// TwinCAT 3 PLC project bnct_plc
// ProgramVersion: 3.1.4024.0
// libraries:
//   Tc2_Standard, * (Beckhoff Automation GmbH)
//   Tc2_System, * (Beckhoff Automation GmbH)
//   Tc3_Module, * (Beckhoff Automation GmbH)
// project tree:
//   DUTs/ Call_Values_To_PC_Struct.TcDUT, Com_StripperEleMach_Struct.TcDUT, ST_FrameCmd.TcDUT
//   DUTs/Read_Status_Struct/ Read_AR_Values_To_PC_Struct.TcDUT, Read_BD_Values_To_PC_Struct.TcDUT, Read_BLPS1_Values_To_PC_Struct.TcDUT, Read_BLPS3_Values_To_PC_Struct.TcDUT, Read_BLVac1_Values_To_PC_Struct.TcDUT, Read_BLVac2_Values_To_PC_Struct.TcDUT, Read_BLVac3_Values_To_PC_Struct.TcDUT, Read_IL_Values_To_PC_Struct.TcDUT, Read_INJLPS_Values_To_PC_Struct.TcDUT, Read_ISPS_Values_To_PC_Struct.TcDUT, Read_ISVac_Values_To_PC_Struct.TcDUT, Read_MainPS_Values_To_PC_Struct.TcDUT, Read_MainVac_Values_To_PC_Struct.TcDUT, Read_RFG_Values_To_PC_Struct.TcDUT, Read_WC_Values_To_PC_Struct.TcDUT
//   DUTs/System_Status_Struct/ S_ARValues_To_PC_Struct.TcDUT, S_BDValues_To_PC_Struct.TcDUT, S_BLPS1Values_To_PC_Struct.TcDUT, S_BLPS3Values_To_PC_Struct.TcDUT, S_BLVac1Values_To_PC_Struct.TcDUT, S_BLVac2Values_To_PC_Struct.TcDUT, S_BLVac3Values_To_PC_Struct.TcDUT, S_ILValues_To_PC_Struct.TcDUT, S_INJLPSValues_To_PC_Struct.TcDUT, S_ISPSValues_To_PC_Struct.TcDUT, S_ISVacValues_To_PC_Struct.TcDUT, S_MainPSValues_To_PC_Struct.TcDUT, S_MainVacValues_To_PC_Struct.TcDUT, S_RFValues_To_PC_Struct.TcDUT, S_WCValues_To_PC_Struct.TcDUT, TCSSys_Struct.TcDUT
//   / PlcTask.TcTTO
//   POUs/ Call_Values_To_PC.TcPOU, Com_StripperEleMach.TcPOU, MAIN.TcPOU, GVL_TCSSys.TcPOU
// real-time tasks:
//   TASK PlcTask: cycle T#10ms, priority 20, ADS port 350

CONFIGURATION bnct_plc
    RESOURCE PLC ON TwinCAT3
        TASK PlcTask(INTERVAL := T#10ms, PRIORITY := 20);
        PROGRAM MAIN WITH PlcTask : MAIN;
        PROGRAM Call_Values_To_PC WITH PlcTask : Call_Values_To_PC;
        PROGRAM Com_StripperEleMach WITH PlcTask : Com_StripperEleMach;
        PROGRAM GVL_TCSSys WITH PlcTask : GVL_TCSSys;
    END_RESOURCE
END_CONFIGURATION

// ---- DUTs/Call_Values_To_PC_Struct.TcDUT
TYPE Call_Values_To_PC_Struct :
UNION
	Read_WC_Values_To_PC:READ_WC_Values_To_PC_Struct; //3.4.1水冷系统
	Read_AR_Values_To_PC:Read_AR_Values_To_PC_Struct; //3.4.2气动系统
	Read_ISVac_Values_To_PC:Read_ISVac_Values_To_PC_Struct; //3.4.3离子源真空系统
	Read_MainVac_Values_To_PC:Read_MainVac_Values_To_PC_Struct; //3.4.4主真空系统
	Read_BLVac1_Values_To_PC:Read_BLVac1_Values_To_PC_Struct; //3.4.5 束流线 1（公共束流线）真空系统
	Read_BLVac2_Values_To_PC:Read_BLVac2_Values_To_PC_Struct; //3.4.6 束流线 2（公共束流线）真空系统
	Read_BLVac3_Values_To_PC:Read_BLVac3_Values_To_PC_Struct; //3.4.7 束流线 3（公共束流线）真空系统
	Read_ISPS_Values_To_PC:Read_ISPS_Values_To_PC_Struct; //3.4.8 离子源电源系统 
	Read_INJLPS_Values_To_PC:Read_INJLPS_Values_To_PC_Struct; //3.4.9 注入线电源系统
	Read_MainPS_Values_To_PC:Read_MainPS_Values_To_PC_Struct;  //3.4.10 主器电源系统
	Read_BLPS1_Values_To_PC:Read_BLPS1_Values_To_PC_Struct; //3.4.11 束流线 1（公共束流线）电源系统
	Read_BLPS3_Values_To_PC:Read_BLPS3_Values_To_PC_Struct; //3.4.12 束流线 3（中子靶束流线）电源系统
	Read_RFG_Values_To_PC:Read_RFG_Values_To_PC_Struct; //3.4.13 高频系统
	Read_BD_Values_To_PC:Read_BD_Values_To_PC_Struct; //3.4.14 束流测量系统
	Read_IL_Values_To_PC:Read_IL_Values_To_PC_Struct; //3.4.15 联锁系统
END_UNION
END_TYPE

// ---- DUTs/Com_StripperEleMach_Struct.TcDUT
TYPE Com_StripperEleMach_Struct :
STRUCT
	Axis1_bEleMachinery_C_Power        : BOOL;
    Axis1_bEleMachinery_C_JF           : BOOL;
    Axis1_bEleMachinery_C_JB           : BOOL;
	Axis1_fEleMachinery_C_AbPos        : REAL;
    Axis1_fEleMachinery_C_AbPosVelo    : REAL;
    Axis1_bEleMachinery_C_AbPosExecute : BOOL;
    Axis1_bEleMachinery_C_Reset        : BOOL;
	Axis2_bEleMachinery_C_Power        : BOOL;
    Axis2_bEleMachinery_C_JF           : BOOL;
    Axis2_bEleMachinery_C_JB           : BOOL;
	Axis2_fEleMachinery_C_AbPos        : REAL;
    Axis2_fEleMachinery_C_AbPosVelo    : REAL;
    Axis2_bEleMachinery_C_AbPosExecute : BOOL;
    Axis2_bEleMachinery_C_Reset        : BOOL;
END_STRUCT
END_TYPE

// ---- DUTs/Read_Status_Struct/Read_AR_Values_To_PC_Struct.TcDUT
TYPE Read_AR_Values_To_PC_Struct :
UNION
	S_ARValues_To_PC:S_ARValues_To_PC_Struct;
END_UNION
END_TYPE

// ---- DUTs/Read_Status_Struct/Read_BD_Values_To_PC_Struct.TcDUT
TYPE Read_BD_Values_To_PC_Struct :
UNION
	S_BDValues_To_PC:S_BDValues_To_PC_Struct;
END_UNION
END_TYPE

// ---- DUTs/Read_Status_Struct/Read_BLPS1_Values_To_PC_Struct.TcDUT
TYPE Read_BLPS1_Values_To_PC_Struct :
UNION
	S_BLPS1Values_To_PC:S_BLPS1Values_To_PC_Struct;
END_UNION
END_TYPE

// ---- DUTs/Read_Status_Struct/Read_BLPS3_Values_To_PC_Struct.TcDUT
TYPE Read_BLPS3_Values_To_PC_Struct :
UNION
	S_BLPS3Values_To_PC:S_BLPS3Values_To_PC_Struct;
END_UNION
END_TYPE

// ---- DUTs/Read_Status_Struct/Read_BLVac1_Values_To_PC_Struct.TcDUT
TYPE Read_BLVac1_Values_To_PC_Struct :
UNION
	S_BLVac1Values_To_PC:S_BLVac1Values_To_PC_Struct;
END_UNION
END_TYPE

// ---- DUTs/Read_Status_Struct/Read_BLVac2_Values_To_PC_Struct.TcDUT
TYPE Read_BLVac2_Values_To_PC_Struct :
UNION
	S_BLVac2Values_To_PC:S_BLVac2Values_To_PC_Struct;
END_UNION
END_TYPE

// ---- DUTs/Read_Status_Struct/Read_BLVac3_Values_To_PC_Struct.TcDUT
TYPE Read_BLVac3_Values_To_PC_Struct :
UNION
	S_BLVac3Values_To_PC:S_BLVac3Values_To_PC_Struct;
END_UNION
END_TYPE

// ---- DUTs/Read_Status_Struct/Read_IL_Values_To_PC_Struct.TcDUT
TYPE Read_IL_Values_To_PC_Struct :
UNION
	S_ILValues_To_PC:S_ILValues_To_PC_Struct;
	// S_ILValues_To_PC:ARRAY[0..116]OF BYTE;
END_UNION
END_TYPE

// ---- DUTs/Read_Status_Struct/Read_INJLPS_Values_To_PC_Struct.TcDUT
TYPE Read_INJLPS_Values_To_PC_Struct :
UNION
	S_INJLPSValues_To_PC:S_INJLPSValues_To_PC_Struct;
END_UNION
END_TYPE

// ---- DUTs/Read_Status_Struct/Read_ISPS_Values_To_PC_Struct.TcDUT
TYPE Read_ISPS_Values_To_PC_Struct :
UNION
	S_ISPSValues_To_PC:S_ISPSValues_To_PC_Struct;
END_UNION
END_TYPE

// ---- DUTs/Read_Status_Struct/Read_ISVac_Values_To_PC_Struct.TcDUT
TYPE Read_ISVac_Values_To_PC_Struct :
UNION
	S_ISVacValues_To_PC:S_ISVacValues_To_PC_Struct;
END_UNION
END_TYPE

// ---- DUTs/Read_Status_Struct/Read_MainPS_Values_To_PC_Struct.TcDUT
TYPE Read_MainPS_Values_To_PC_Struct :
UNION
	S_MainPSValues_To_PC:S_MainPSValues_To_PC_Struct;
END_UNION
END_TYPE

// ---- DUTs/Read_Status_Struct/Read_MainVac_Values_To_PC_Struct.TcDUT
TYPE Read_MainVac_Values_To_PC_Struct :
UNION
	S_MainVacValues_To_PC:S_MainVacValues_To_PC_Struct;
END_UNION
END_TYPE

// ---- DUTs/Read_Status_Struct/Read_RFG_Values_To_PC_Struct.TcDUT
TYPE Read_RFG_Values_To_PC_Struct :
UNION
	S_RFValues_To_PC:S_RFValues_To_PC_Struct;
END_UNION
END_TYPE

// ---- DUTs/Read_Status_Struct/Read_WC_Values_To_PC_Struct.TcDUT
TYPE Read_WC_Values_To_PC_Struct :
UNION
	S_WCValues_To_PC:S_WCValues_To_PC_Struct;
END_UNION
END_TYPE

// ---- DUTs/System_Status_Struct/S_ARValues_To_PC_Struct.TcDUT
TYPE S_ARValues_To_PC_Struct :
STRUCT
	PARAM000:BOOL ; //注入线隔断阀开到位
	PARAM001:BOOL ; //注入线隔断阀关到位
	PARAM002:BOOL ; //注入线隔断阀正在开
	PARAM003:BOOL ; //注入线隔断阀正在关
	PARAM004:BOOL ; //注入线隔断阀开启操作错误
	PARAM005:BOOL ; //注入线隔断阀关闭操作错误
	PARAM006:BOOL ; //束流线隔断阀 1 开到位
	PARAM007:BOOL ; //束流线隔断阀 1 关到位
	PARAM008:BOOL ; //束流线隔断阀 1 正在开
	PARAM009:BOOL ; //束流线隔断阀 1 正在关
	PARAM010:BOOL ; //束流线隔断阀 1 开启操作错误
	PARAM011:BOOL ; //束流线隔断阀 1 关闭操作错误
	PARAM012:BOOL ; //束流线隔断阀 2 开到位
	PARAM013:BOOL ; //束流线隔断阀 2 关到位
	PARAM014:BOOL ; //束流线隔断阀 2 正在开
	PARAM015:BOOL ; //束流线隔断阀 2 正在关
	PARAM016:BOOL ; //束流线隔断阀 2 开启操作错误
	PARAM017:BOOL ; //束流线隔断阀 2 关闭操作错误
	PARAM018:BOOL ; //束流线隔断阀 3 开到位
	PARAM019:BOOL ; //束流线隔断阀 3 关到位
	PARAM020:BOOL ; //束流线隔断阀 3 正在开
	PARAM021:BOOL ; //束流线隔断阀 3 正在关
	PARAM022:BOOL ; //束流线隔断阀 3 开启操作错误
	PARAM023:BOOL ; //束流线隔断阀 3 关闭操作错误
	PARAM024:BOOL ; //注入线 FC 拉出到位
	PARAM025:BOOL ; //注入线 FC 插入到位
	PARAM026:BOOL ; //注入线 FC 正在拉出
	PARAM027:BOOL ; //注入线 FC 正在插入
	PARAM028:BOOL ; //注入线 FC 拉出操作错误
	PARAM029:BOOL ; //注入线 FC 插入操作错误
	PARAM030:BOOL ; //内靶拉出到位
	PARAM031:BOOL ; //内靶插入到位
	PARAM032:BOOL ; //内靶正在拉出
	PARAM033:BOOL ; //内靶正在插入
	PARAM034:BOOL ; //内靶拉出操作错误
	PARAM035:BOOL ; //内靶插入操作错误
	PARAM036:BOOL ; //引出 FC 拉出到位
	PARAM037:BOOL ; //引出 FC 插入到位
	PARAM038:BOOL ; //引出 FC 正在拉出
	PARAM039:BOOL ; //引出 FC 正在插入
	PARAM040:BOOL ; //引出 FC 拉出操作错误
	PARAM041:BOOL ; //引出 FC 插入操作错误
	PARAM042:BOOL ; //荧光靶 1 拉出到位
	PARAM043:BOOL ; //荧光靶 1 插入到位
	PARAM044:BOOL ; //荧光靶 1 正在拉出
	PARAM045:BOOL ; //荧光靶 1 正在插入
	PARAM046:BOOL ; //荧光靶 1 拉出操作错误
	PARAM047:BOOL ; //荧光靶 1 插入操作错误
	PARAM048:BOOL ; //荧光靶 2 拉出到位
	PARAM049:BOOL ; //荧光靶 2 插入到位
	PARAM050:BOOL ; //荧光靶 2 正在拉出
	PARAM051:BOOL ; //荧光靶 2 正在插入
	PARAM052:BOOL ; //荧光靶 2 拉出操作错误
	PARAM053:BOOL ; //荧光靶 2 插入操作错误
	PARAM054:BOOL ; //荧光靶 3 拉出到位
	PARAM055:BOOL ; //荧光靶 3 插入到位
	PARAM056:BOOL ; //荧光靶 3 正在拉出
	PARAM057:BOOL ; //荧光靶 3 正在插入
	PARAM058:BOOL ; //荧光靶 3 拉出操作错误
	PARAM059:BOOL ; //荧光靶 3 插入操作错误
	PARAM060:BOOL ; //双丝 1 拉出到位
	PARAM061:BOOL ; //双丝 1 插入到位
	PARAM062:BOOL ; //双丝 1 正在拉出
	PARAM063:BOOL ; //双丝 1 正在插入
	PARAM064:BOOL ; //双丝 1 拉出操作错误
	PARAM065:BOOL ; //双丝 1 插入操作错误
	PARAM066:BOOL ; //双丝 2 拉出到位
	PARAM067:BOOL ; //双丝 2 插入到位
	PARAM068:BOOL ; //双丝 2 正在拉出
	PARAM069:BOOL ; //双丝 2 正在插入
	PARAM070:BOOL ; //双丝 2 拉出操作错误
	PARAM071:BOOL ; //双丝 2 插入操作错误

END_STRUCT
END_TYPE

// ---- DUTs/System_Status_Struct/S_BDValues_To_PC_Struct.TcDUT
TYPE S_BDValues_To_PC_Struct :
STRUCT
	PARAM000:BOOL  ;// 剥离靶1电机使能指令 
	PARAM001:BOOL  ;// 剥离靶1电机绝对运动触发指令 
	PARAM002:REAL  ;// 剥离靶1电机绝对运动位置指令 
	PARAM003:REAL  ;// 剥离靶1电机绝对运动速度指令 
	PARAM004:BOOL  ;// 剥离靶1电机复位指令 
	PARAM005:BOOL  ;// 剥离靶1电机JOG前进指令 
	PARAM006:BOOL  ;// 剥离靶1电机JOG后退指令 
	PARAM007:BOOL  ;// 剥离靶1电机急停指令 
	PARAM008:BOOL  ;// 剥离靶1电机绝对运动完成 
	PARAM009:BOOL  ;// 剥离靶1电机绝对运动正在进行 
	PARAM010:REAL  ;// 剥离靶1电机位置状态 
	PARAM011:REAL  ;// 剥离靶1电机速度状态 
	PARAM012:BOOL  ;// 剥离靶1电机JOG运动完成 
	PARAM013:BOOL  ;// 剥离靶1电机JOG运动正在进行 
	PARAM014:UDINT ;// 剥离靶1电机故障编码 
	PARAM015:INT   ;// 剥离靶1电位器位置 
	PARAM016:BOOL  ;// 剥离靶2电机使能指令 
	PARAM017:BOOL  ;// 剥离靶2电机绝对运动触发指令 
	PARAM018:REAL  ;// 剥离靶2电机绝对运动位置指令 
	PARAM019:REAL  ;// 剥离靶2电机绝对运动速度指令 
	PARAM020:BOOL  ;// 剥离靶2电机复位指令 
	PARAM021:BOOL  ;// 剥离靶2电机JOG前进指令 
	PARAM022:BOOL  ;// 剥离靶2电机JOG后退指令 
	PARAM023:BOOL  ;// 剥离靶2电机急停指令 
	PARAM024:BOOL  ;// 剥离靶2电机绝对运动完成 
	PARAM025:BOOL  ;// 剥离靶2电机绝对运动正在进行 
	PARAM026:REAL  ;// 剥离靶2电机位置 
	PARAM027:REAL  ;// 剥离靶2电机速度 
	PARAM028:BOOL  ;// 剥离靶2电机JOG运动完成 
	PARAM029:BOOL  ;// 剥离靶2电机JOG运动正在进行 
	PARAM030:UDINT ;// 剥离靶2电机故障编码
	PARAM031:INT   ;// 剥离靶2电位器位置 
	PARAM032:REAL  ;// 束流通道1（mA）：注入FC 
	PARAM033:REAL  ;// 束流通道2（mA）:内靶 
	PARAM034:REAL  ;// 束流通道3（mA）：剥离靶 
	PARAM035:REAL  ;// 束流通道4（mA）：引出FC 
	PARAM036:REAL  ;// 束流通道5（mA）：铍靶 
	PARAM037:REAL  ;// 束流通道6（uA）：备用1 
	PARAM038:REAL  ;// 束流通道7（uA）：备用2 
	PARAM039:REAL  ;// 束流通道8（mA）：备用3 
	PARAM040:REAL  ;// 束流通道9（uA）：光阑1-上 
	PARAM041:REAL  ;// 束流通道10（uA）：光阑2-上 
	PARAM042:REAL  ;// 束流通道11（uA）：光阑1-下 
	PARAM043:REAL  ;// 束流通道12（uA）：光阑2-下 
	PARAM044:REAL  ;// 束流通道13（uA）：光阑1-左 
	PARAM045:REAL  ;// 束流通道14（uA）：光阑2-左 
	PARAM046:REAL  ;// 束流通道15（uA）：光阑1-右 
	PARAM047:REAL  ;// 束流通道16（uA）：光阑2-右 
END_STRUCT
END_TYPE

// ---- DUTs/System_Status_Struct/S_BLPS1Values_To_PC_Struct.TcDUT
TYPE S_BLPS1Values_To_PC_Struct :
STRUCT
	PARAM000:BOOL ; //  束流线1电源自动运行，TRUE为开启 
	PARAM001:REAL ; //  四级透镜1电源电流设置值（A） 
	PARAM002:BOOL ; //  四级透镜1电源已开 
	PARAM003:BOOL ; //  四级透镜1电源已关 
	PARAM004:BOOL ; //  四级透镜1电源正在开 
	PARAM005:BOOL ; //  四级透镜1电源正在关 
	PARAM006:REAL ; //  四级透镜1电源运行电流（A） 
	PARAM007:REAL ; //  四级透镜1电源运行电压（V） 
	PARAM008:BOOL ; //  TRUE时四级透镜1电源故障 
	PARAM009:BOOL ; //  TRUE时四级透镜1电源电流操作错误 
	PARAM010:REAL ; //  XY1-X导向电源电流设置值（A） 
	PARAM011:BOOL ; //  XY1-X导向电源已开 
	PARAM012:BOOL ; //  XY1-X导向电源已关 
	PARAM013:BOOL ; //  XY1-X导向电源正在开 
	PARAM014:BOOL ; //  XY1-X导向电源正在关 
	PARAM015:REAL ; //  XY1-X导向电源运行电流（A） 
	PARAM016:REAL ; //  XY1-X导向电源运行电压（V） 
	PARAM017:BOOL ; //  TRUE时XY1-X导向电源故障 
	PARAM018:BOOL ; //  TRUE时XY1-X电源电流操作错误 
	PARAM019:BOOL ; //  TRUE时XY1-X导向电源通讯正常 
	PARAM020:REAL ; //  XY1-Y导向电源电流设置值（A） 
	PARAM021:BOOL ; //  XY1-Y导向电源已开 
	PARAM022:BOOL ; //  XY1-Y导向电源已关 
	PARAM023:BOOL ; //  XY1-Y导向电源正在开 
	PARAM024:BOOL ; //  XY1-Y导向电源正在关 
	PARAM025:REAL ; //  XY1-Y导向电源运行电流（A） 
	PARAM026:REAL ; //  XY1-Y导向电源运行电压（V） 
	PARAM027:BOOL ; //  TRUE时XY1-Y导向电源故障 
	PARAM028:BOOL ; //  TRUE时XY1-Y电源电流操作错误 
	PARAM029:BOOL ; //  TRUE时XY1-Y导向电源通讯正常 
	PARAM030:REAL ; //  四极透镜2电源电流设置值（A） 
	PARAM031:BOOL ; //  四极透镜2电源已开 
	PARAM032:BOOL ; //  四极透镜2电源已关 
	PARAM033:BOOL ; //  四极透镜2电源正在开 
	PARAM034:BOOL ; //  四极透镜2电源正在关 
	PARAM035:REAL ; //  四极透镜2电源运行电流（A） 
	PARAM036:REAL ; //  四极透镜2电源运行电压（V） 
	PARAM037:BOOL ; //  TRUE时四极透镜2电源故障
	PARAM038:BOOL ; //  TRUE时四极透镜2电源电流操作错误 
	PARAM039:REAL ; //  四极透镜3电源电流设置值（A） 
	PARAM040:BOOL ; //  四极透镜3电源已开 
	PARAM041:BOOL ; //  四极透镜3电源已关 
	PARAM042:BOOL ; //  四极透镜3电源正在开 
	PARAM043:BOOL ; //  四极透镜3电源正在关 
	PARAM044:REAL ; //  四极透镜3电源运行电流（A） 
	PARAM045:REAL ; //  四极透镜3电源运行电压（V） 
	PARAM046:BOOL ; //  TRUE时四极透镜3电源故障 
	PARAM047:BOOL ; //  TRUE时四极透镜3电源电流操作错误 
	PARAM048:REAL ; //  偏转磁铁电源电流设置值（A） 
	PARAM049:BOOL ; //  偏转磁铁电源已开 
	PARAM050:BOOL ; //  偏转磁铁电源已关 
	PARAM051:BOOL ; //  偏转磁铁电源正在开 
	PARAM052:BOOL ; //  偏转磁铁电源正在关 
	PARAM053:REAL ; //  偏转磁铁电源运行电流（A） 
	PARAM054:REAL ; //  偏转磁铁电源运行电压（V） 
	PARAM055:BOOL ; //  TRUE时偏转磁铁电源故障 
	PARAM056:BOOL ; //  TRUE时偏转磁铁电源电流操作错误 
	PARAM057:REAL ; //  四八级1-1电源电流设置值（A） 
	PARAM058:BOOL ; //  四八级1-1电源已开 
	PARAM059:BOOL ; //  四八级1-1电源已关 
	PARAM060:BOOL ; //  四八级1-1电源正在开 
	PARAM061:BOOL ; //  四八级1-1电源正在关 
	PARAM062:REAL ; //  四八级1-1电源运行电流（A） 
	PARAM063:REAL ; //  四八级1-1电源运行电压（V） 
	PARAM064:BOOL ; //  TRUE时四八级1-1电源故障 
	PARAM065:BOOL ; //  TRUE时四八级1-1电源电流操作错误
	PARAM066:REAL ; //  四八级1-2电源电流设置值（A） 
	PARAM067:BOOL ; //  四八级1-2电源已开 
	PARAM068:BOOL ; //  四八级1-2电源已关 
	PARAM069:BOOL ; //  四八级1-2电源正在开 
	PARAM070:BOOL ; //  四八级1-2电源正在关 
	PARAM071:REAL ; //  四八级1-2电源运行电流（A） 
	PARAM072:REAL ; //  四八级1-2电源运行电压（V） 
	PARAM073:BOOL ; //  TRUE时四八级1-2电源故障 
	PARAM074:BOOL ; //  TRUE时四八级1-2电源电流操作错误 
	PARAM075:REAL ; //  四八级2-1电源电流设置值（A） 
	PARAM076:BOOL ; //  四八级2-1电源已开 
	PARAM077:BOOL ; //  四八级2-1电源已关 
	PARAM078:BOOL ; //  四八级2-1电源正在开 
	PARAM079:BOOL ; //  四八级2-1电源正在关 
	PARAM080:REAL ; //  四八级2-1电源运行电流（A） 
	PARAM081:REAL ; //  四八级2-1电源运行电压（V） 
	PARAM082:BOOL ; //  TRUE时四八级2-1电源故障 
	PARAM083:BOOL ; //  TRUE时四八级2-1电源电流操作错误 
	PARAM084:REAL ; //  四八级2-2电源电流设置值（A） 
	PARAM085:BOOL ; //  四八级2-2电源已开 
	PARAM086:BOOL ; //  四八级2-2电源已关 
	PARAM087:BOOL ; //  四八级2-2电源正在开 
	PARAM088:BOOL ; //  四八级2-2电源正在关 
	PARAM089:REAL ; //  四八级2-2电源运行电流（A） 
	PARAM090:REAL ; //  四八级2-2电源运行电压（V） 
	PARAM091:BOOL ; //  TRUE时四八级2-2电源故障 
	PARAM092:BOOL ; //  TRUE时四八级2-2电源电流操作错误 
	PARAM093:BOOL ; //  引出FC抑制偏压电源已开 
	PARAM094:BOOL ; //  引出FC抑制偏压电源已关 
	PARAM095:BOOL ; //  引出FC抑制偏压电源正在开 
	PARAM096:BOOL ; //  引出FC抑制偏压电源正在关 
	PARAM097:REAL ; //  引出FC抑制偏压电源运行电流（A） 
	PARAM098:REAL ; //  引出FC抑制偏压电源运行电压（V） 
	PARAM099:BOOL ; //  Ture为引出FC抑制偏压电源故障 
	PARAM100:BOOL ; //  Ture为引出FC抑制偏压电源远控 
	PARAM101:BOOL ; //  引出FC抑制偏压电源正极 
	PARAM102:BOOL ; //  引出FC抑制偏压电源负极 
	PARAM103:BOOL ; //  引出FC抑制偏压电源电压操作错误 

END_STRUCT
END_TYPE

// ---- DUTs/System_Status_Struct/S_BLPS3Values_To_PC_Struct.TcDUT
TYPE S_BLPS3Values_To_PC_Struct :
STRUCT
	PARAM000:BOOL ;// 束流线3电源自动运行，TRUE为开启 
	PARAM001:REAL ;// 四级透镜4电源电流设置值（A） 
	PARAM002:BOOL ;// 四级透镜4电源已开 
	PARAM003:BOOL ;// 四级透镜4电源已关 
	PARAM004:BOOL ;// 四级透镜4电源正在开 
	PARAM005:BOOL ;// 四级透镜4电源正在关 
	PARAM006:REAL ;// 四级透镜4电源运行电流（A） 
	PARAM007:REAL ;// 四级透镜4电源运行电压（V） 
	PARAM008:BOOL ;// TRUE时四级透镜4电源故障 
	PARAM009:BOOL ;// 四级透镜4电源电流操作故障 
	PARAM010:REAL ;// 四八级3-1电源电流设置值（A） 
	PARAM011:BOOL ;// 四八级3-1电源已开
	PARAM012:BOOL ;// 四八级3-1电源已关 
	PARAM013:BOOL ;// 四八级3-1电源正在开 
	PARAM014:BOOL ;// 四八级3-1电源正在关 
	PARAM015:REAL ;// 四八级3-1电源运行电流（A） 
	PARAM016:REAL ;// 四八级3-1电源运行电压（V） 
	PARAM017:BOOL ;// TRUE时四八级3-1电源故障 
	PARAM018:BOOL ;// 四八级3-1电源电流操作错误 
	PARAM019:REAL ;// 四八级3-2电源电流设置值（A） 
	PARAM020:BOOL ;// 四八级3-2电源已开 
	PARAM021:BOOL ;// 四八级3-2电源已关 
	PARAM022:BOOL ;// 四八级3-2电源正在开 
	PARAM023:BOOL ;// 四八级3-2电源正在关 
	PARAM024:REAL ;// 四八级3-2电源运行电流（A） 
	PARAM025:REAL ;// 四八级3-2电源运行电压（V） 
	PARAM026:BOOL ;// TRUE时四八级3-2电源故障 
	PARAM027:BOOL ;// 四八级3-2电源电流操作错误 
	PARAM028:BOOL ;// 双丝抑制偏压电源已开 
	PARAM029:BOOL ;// 双丝抑制偏压电源已关 
	PARAM030:BOOL ;// 双丝抑制偏压电源正在开 
	PARAM031:BOOL ;// 双丝抑制偏压电源正在关 
	PARAM032:REAL ;// 双丝抑制偏压电源运行电流（A） 
	PARAM033:REAL ;// 双丝抑制偏压电源运行电压（V） 
	PARAM034:BOOL ;// Ture为双丝抑制偏压电源故障 
	PARAM035:BOOL ;// Ture为双丝抑制偏压电源远控 
	PARAM036:BOOL ;// 双丝抑制偏压电源正极 
	PARAM037:BOOL ;// 双丝抑制偏压电源负极 
	PARAM038:BOOL ;// 双丝抑制偏压电源电压操作错误 

END_STRUCT
END_TYPE

// ---- DUTs/System_Status_Struct/S_BLVac1Values_To_PC_Struct.TcDUT
TYPE S_BLVac1Values_To_PC_Struct :
STRUCT
	PARAM000:BOOL ; // 束流线1低真空自动运行，True代表开 
	PARAM001:BOOL ; // 束流线1高真空自动运行，True代表开 
	PARAM002:BOOL ; // 束流线角阀1开到位 
	PARAM003:BOOL ; // 束流线角阀1关到位 
	PARAM004:BOOL ; // 束流线角阀1正在开 
	PARAM005:BOOL ; // 束流线角阀1正在关 
	PARAM006:BOOL ; // 束流线角阀1开启操作错误 
	PARAM007:BOOL ; // 束流线角阀1关闭操作错误 
	PARAM008:BOOL ; // 束流线放气阀1开到位 
	PARAM009:BOOL ; // 束流线放气阀1关到位 
	PARAM010:BOOL ; // 束流线放气阀1正在开 
	PARAM011:BOOL ; // 束流线放气阀1正在关 
	PARAM012:BOOL ; // 束流线放气阀1开启操作错误 
	PARAM013:BOOL ; // 束流线放气阀1关闭操作错误 
	PARAM014:BOOL ; // 束流线1机械泵开到位 
	PARAM015:BOOL ; // 束流线1机械泵关到位 
	PARAM016:BOOL ; // 束流线1机械泵正在开 
	PARAM017:BOOL ; // 束流线1机械泵正在关 
	PARAM018:BOOL ; // 束流线1机械泵开启操作错误 
	PARAM019:BOOL ; // 束流线1机械泵关闭操作错误 
	PARAM020:BOOL ; // 束流线1分子泵V5达到频率值 
	PARAM021:BOOL ; // 束流线1分子泵V5频率下降到0 
	PARAM022:BOOL ; // 束流线1分子泵V5故障 
	PARAM023:BOOL ; // 束流线1分子泵V5频率上升中 
	PARAM024:BOOL ; // 束流线1分子泵V5频率下降中 
	PARAM025:BOOL ; // 束流线1分子泵V5开启操作错误 
	PARAM026:BOOL ; // 束流线1分子泵V5关闭操作错误 
	PARAM027:REAL ; // 束流线1分子泵V5输出频率（Hz） 
	PARAM028:LREAL ; // 束流线1低真空度（mbar） 
	PARAM029:LREAL ; // 束流线1高真空度（mbar） 
	PARAM030:BOOL ; // 束流线1低真空已达标 
	PARAM031:BOOL ; // 束流线1高真空已达标 
END_STRUCT
END_TYPE

// ---- DUTs/System_Status_Struct/S_BLVac2Values_To_PC_Struct.TcDUT
TYPE S_BLVac2Values_To_PC_Struct :
STRUCT
	PARAM000:BOOL ; // 束流线2低真空自动运行，True代表开 
	PARAM001:BOOL ; // 束流线2高真空自动运行，True代表开 
	PARAM002:BOOL ; // 束流线角阀2开到位 
	PARAM003:BOOL ; // 束流线角阀2关到位 
	PARAM004:BOOL ; // 束流线角阀2正在开 
	PARAM005:BOOL ; // 束流线角阀2正在关 
	PARAM006:BOOL ; // 束流线角阀2开启操作错误 
	PARAM007:BOOL ; // 束流线角阀2关闭操作错误 
	PARAM008:BOOL ; // 束流线放气阀2开到位 
	PARAM009:BOOL ; // 束流线放气阀2关到位 
	PARAM010:BOOL ; // 束流线放气阀2正在开 
	PARAM011:BOOL ; // 束流线放气阀2正在关 
	PARAM012:BOOL ; // 束流线放气阀2开启操作错误 
	PARAM013:BOOL ; // 束流线放气阀2关闭操作错误 
	PARAM014:BOOL ; // 束流线2机械泵开到位 
	PARAM015:BOOL ; // 束流线2机械泵关到位
	PARAM016:BOOL ; // 束流线2机械泵正在开 
	PARAM017:BOOL ; // 束流线2机械泵正在关 
	PARAM018:BOOL ; // 束流线2机械泵开启操作错误 
	PARAM019:BOOL ; // 束流线2机械泵关闭操作错误 
	PARAM020:BOOL ; // 束流线2分子泵V6达到频率值 
	PARAM021:BOOL ; // 束流线2分子泵V6频率下降到0 
	PARAM022:BOOL ; // 束流线2分子泵V6故障 
	PARAM023:BOOL ; // 束流线2分子泵V6频率上升中 
	PARAM024:BOOL ; // 束流线2分子泵V6频率下降中 
	PARAM025:BOOL ; // 束流线2分子泵V6开启操作错误 
	PARAM026:BOOL ; // 束流线2分子泵V6关闭操作错误 
	PARAM027:REAL ; // 束流线2分子泵V6输出频率（Hz） 
	PARAM028:LREAL ; // 束流线2低真空度（mbar） 
	PARAM029:LREAL ; // 束流线2高真空度（mbar） 
	PARAM030:BOOL ; // 束流线2低真空已达标 
	PARAM031:BOOL ; // 束流线2高真空已达标
END_STRUCT
END_TYPE

// ---- DUTs/System_Status_Struct/S_BLVac3Values_To_PC_Struct.TcDUT
TYPE S_BLVac3Values_To_PC_Struct :
STRUCT
	PARAM000:BOOL ; // 束流线3低真空自动运行，True代表开 
	PARAM001:BOOL ; // 束流线3高真空自动运行，True代表开 
	PARAM002:BOOL ; // 束流线角阀3开到位 
	PARAM003:BOOL ; // 束流线角阀3关到位 
	PARAM004:BOOL ; // 束流线角阀3正在开 
	PARAM005:BOOL ; // 束流线角阀3正在关
	PARAM006:BOOL ; // 束流线角阀3开启操作错误 
	PARAM007:BOOL ; // 束流线角阀3关闭操作错误 
	PARAM008:BOOL ; // 束流线放气阀3开到位 
	PARAM009:BOOL ; // 束流线放气阀3关到位 
	PARAM010:BOOL ; // 束流线放气阀3正在开 
	PARAM011:BOOL ; // 束流线放气阀3正在关 
	PARAM012:BOOL ; // 束流线放气阀3开启操作错误 
	PARAM013:BOOL ; // 束流线放气阀2关闭操作错误 
	PARAM014:BOOL ; // 束流线3机械泵开到位 
	PARAM015:BOOL ; // 束流线3机械泵关到位 
	PARAM016:BOOL ; // 束流线3机械泵正在开 
	PARAM017:BOOL ; // 束流线3机械泵正在关 
	PARAM018:BOOL ; // 束流线3机械泵开启操作错误 
	PARAM019:BOOL ; // 束流线3机械泵关闭操作错误 
	PARAM020:BOOL ; // 束流线3分子泵V7达到频率值 
	PARAM021:BOOL ; // 束流线3分子泵V7频率下降到0 
	PARAM022:BOOL ; // 束流线3分子泵V7故障 
	PARAM023:BOOL ; // 束流线3分子泵V7频率上升中 
	PARAM024:BOOL ; // 束流线3分子泵V7频率下降中 
	PARAM025:BOOL ; // 束流线3分子泵V7开启操作错误 
	PARAM026:BOOL ; // 束流线3分子泵V7关闭操作错误 
	PARAM027:REAL ; // 束流线3分子泵V7输出频率（Hz） 
	PARAM028:LREAL ; // 束流线3低真空度（mbar） 
	PARAM029:LREAL ; // 束流线3高真空度（mbar） 
	PARAM030:BOOL ; // 束流线3低真空已达标 
	PARAM031:BOOL ; // 束流线3高真空已达标 
END_STRUCT
END_TYPE

// ---- DUTs/System_Status_Struct/S_ILValues_To_PC_Struct.TcDUT
TYPE S_ILValues_To_PC_Struct :
STRUCT
	PARAM000:REAL ;// 注入线法拉第筒温度节点01（℃） 
	PARAM001:REAL ;// 内靶温度节点02（℃） 
	PARAM002:REAL ;// 引出法拉第筒温度节点03（℃） 
	PARAM003:REAL ;// 温度节点04（℃） 
	PARAM004:REAL ;// 温度节点05（℃）
	PARAM005:REAL ;// 温度节点06（℃） 
	PARAM006:REAL ;// 温度节点07（℃） 
	PARAM007:REAL ;// 温度节点08（℃） 
	PARAM008:BOOL ;// 已经移去接地 
	PARAM009:BOOL ;// 地坑栅栏门已经关闭 
	PARAM010:BOOL ;// 加速器已合盖 
	PARAM011:BOOL ;// 无源节点01 
	PARAM012:BOOL ;// 无源节点02 
	PARAM013:BOOL ;// 离子源角阀2联锁开 
	PARAM014:BOOL ;// 离子源角阀2联锁关 
	PARAM015:BOOL ;// 注入线放气阀联锁开 
	PARAM016:BOOL ;// 注入线放气阀联锁关 
	PARAM017:BOOL ;// 离子源干泵联锁开 
	PARAM018:BOOL ;// 离子源干泵联锁关 
	PARAM019:BOOL ;// 离子源分子泵V1联锁开 
	PARAM020:BOOL ;// 离子源分子泵V1联锁关 
	PARAM021:BOOL ;// 离子源分子泵V3联锁开 
	PARAM022:BOOL ;// 离子源分子泵V3联锁关 
	PARAM023:BOOL ;// 离子源分子泵V4联锁开 
	PARAM024:BOOL ;// 离子源分子泵V4联锁关 
	PARAM025:BOOL ;// 冷泵隔断阀1联锁开 
	PARAM026:BOOL ;// 冷泵隔断阀1联锁关 
	PARAM027:BOOL ;// 冷泵隔断阀2联锁开 
	PARAM028:BOOL ;// 冷泵隔断阀2联锁关 
	PARAM029:BOOL ;// 主真空角阀1联锁开 
	PARAM030:BOOL ;// 主真空角阀1联锁关 
	PARAM031:BOOL ;// 主真空放气阀联锁开 
	PARAM032:BOOL ;// 主真空放气阀联锁关
	PARAM033:BOOL ;// 主真空干泵联锁开 
	PARAM034:BOOL ;// 主真空干泵联锁关 
	PARAM035:BOOL ;// 主真空分子泵V2联锁开 
	PARAM036:BOOL ;// 主真空分子泵V2联锁关 
	PARAM037:BOOL ;// 冷泵前级阀1联锁开 
	PARAM038:BOOL ;// 冷泵前级阀1联锁关 
	PARAM039:BOOL ;// 冷泵1联锁开 
	PARAM040:BOOL ;// 冷泵1联锁关 
	PARAM041:BOOL ;// 冷泵前级阀2联锁开 
	PARAM042:BOOL ;// 冷泵前级阀2联锁关 
	PARAM043:BOOL ;// 冷泵2联锁开 
	PARAM044:BOOL ;// 冷泵2联锁关 
	PARAM045:BOOL ;// 束流线1角阀联锁开 
	PARAM046:BOOL ;// 束流线1角阀联锁关 
	PARAM047:BOOL ;// 束流线1放气阀联锁开 
	PARAM048:BOOL ;// 束流线1放气阀联锁关 
	PARAM049:BOOL ;// 束流线1干泵联锁开 
	PARAM050:BOOL ;// 束流线1干泵联锁关 
	PARAM051:BOOL ;// 束流线1分子泵V5联锁开 
	PARAM052:BOOL ;// 束流线1分子泵V5联锁关 
	PARAM053:BOOL ;// 束流线2角阀联锁开 
	PARAM054:BOOL ;// 束流线2角阀联锁关 
	PARAM055:BOOL ;// 束流线2放气阀联锁开 
	PARAM056:BOOL ;// 束流线2放气阀联锁关 
	PARAM057:BOOL ;// 束流线2干泵联锁开 
	PARAM058:BOOL ;// 束流线2干泵联锁关 
	PARAM059:BOOL ;// 束流线2分子泵V6联锁开 
	PARAM060:BOOL ;// 束流线2分子泵V6联锁关
	PARAM061:BOOL ;// 束流线3角阀联锁开 
	PARAM062:BOOL ;// 束流线3角阀联锁关 
	PARAM063:BOOL ;// 束流线3放气阀联锁开 
	PARAM064:BOOL ;// 束流线3放气阀联锁关 
	PARAM065:BOOL ;// 束流线3干泵联锁开 
	PARAM066:BOOL ;// 束流线3干泵联锁关 
	PARAM067:BOOL ;// 束流线3分子泵V7联锁开 
	PARAM068:BOOL ;// 束流线3分子泵V7联锁关 
	PARAM069:BOOL ;// 注入线隔断阀联锁拉开 
	PARAM070:BOOL ;// 注入线隔断阀联锁插入 
	PARAM071:BOOL ;// 注入线法拉第筒联锁拉开 
	PARAM072:BOOL ;// 注入线法拉第筒联锁插入 
	PARAM073:BOOL ;// 内靶联锁拉开 
	PARAM074:BOOL ;// 内靶联锁插入 
	PARAM075:BOOL ;// 束流线1隔断阀联锁开 
	PARAM076:BOOL ;// 束流线1隔断阀联锁关 
	PARAM077:BOOL ;// 束流线2隔断阀联锁开 
	PARAM078:BOOL ;// 束流线2隔断阀联锁关 
	PARAM079:BOOL ;// 束流线3隔断阀联锁开 
	PARAM080:BOOL ;// 束流线3隔断阀联锁关 
	PARAM081:BOOL ;// 引出法拉第筒联锁拉开 
	PARAM082:BOOL ;// 引出法拉第筒联锁插入 
	PARAM083:BOOL ;// 离子源高压电源联锁开 
	PARAM084:BOOL ;// 离子源高压电源联锁关 
	PARAM085:BOOL ;// 正偏转版电源联锁开 
	PARAM086:BOOL ;// 正偏转版电源联锁关 
	PARAM087:BOOL ;// 负偏转版电源联锁开 
	PARAM088:BOOL ;// 正偏转版电源联锁关 
END_STRUCT
END_TYPE

// ---- DUTs/System_Status_Struct/S_INJLPSValues_To_PC_Struct.TcDUT
TYPE S_INJLPSValues_To_PC_Struct :
STRUCT
	PARAM000:BOOL ; // 注入线电源系统自动运行，TRUE为开启 
	PARAM001:REAL ; // XY1-X导向电源电流设置值（A） 
	PARAM002:BOOL ; // XY1-X导向电源已开 
	PARAM003:BOOL ; // XY1-X导向电源已关 
	PARAM004:BOOL ; // XY1-X导向电源正在开 
	PARAM005:BOOL ; // XY1-X导向电源正在关 
	PARAM006:REAL ; // XY1-X导向电源运行电流（A） 
	PARAM007:REAL ; // XY1-X导向电源运行电压（V） 
	PARAM008:BOOL ; // TRUE时XY1-X导向电源故障 
	PARAM009:BOOL ; // TRUE时XY1-X导向电源电流操作错误
	PARAM010:BOOL ; // TRUE时XY1-X导向电源通讯正常 
	PARAM011:REAL ; // XY1-Y导向电源电流设置值（A） 
	PARAM012:BOOL ; // XY1-Y导向电源已开 
	PARAM013:BOOL ; // XY1-Y导向电源已关 
	PARAM014:BOOL ; // XY1-Y导向电源正在开 
	PARAM015:BOOL ; // XY1-Y导向电源正在关 
	PARAM016:REAL ; // XY1-Y导向电源运行电流（A） 
	PARAM017:REAL ; // XY1-Y导向电源运行电压（V） 
	PARAM018:BOOL ; // TRUE时XY1-Y导向电源故障 
	PARAM019:BOOL ; // TRUE时XY1-Y导向电源通讯正常 
	PARAM020:BOOL ; // TRUE时XY1-Y导向电源电流操作错误 
	PARAM021:REAL ; // 螺旋管1电源电流设置值（A） 
	PARAM022:BOOL ; // 螺旋管1电源已开 
	PARAM023:BOOL ; // 螺旋管1电源已关 
	PARAM024:BOOL ; // 螺旋管1电源正在开 
	PARAM025:BOOL ; // 螺旋管1电源正在关 
	PARAM026:REAL ; // 螺旋管1电源运行电流（A） 
	PARAM027:REAL ; // 螺旋管1电源运行电压（V） 
	PARAM028:BOOL ; // TRUE时螺旋管1电源故障 
	PARAM029:BOOL ; // TRUE时螺旋管1电源电流操作错误 
	PARAM030:REAL ; // XY2-X导向电源电流设置值（A） 
	PARAM031:BOOL ; // XY2-X导向电源已开 
	PARAM032:BOOL ; // XY2-X导向电源已关 
	PARAM033:BOOL ; // XY2-X导向电源正在开 
	PARAM034:BOOL ; // XY2-X导向电源正在关 
	PARAM035:REAL ; // XY2-X导向电源运行电流（A） 
	PARAM036:REAL ; // XY2-X导向电源运行电压（V） 
	PARAM037:BOOL ; // TRUE时XY2-X导向电源故障 
	PARAM038:BOOL ; // TRUE时XY2-X导向电源电流操作错误 
	PARAM039:BOOL ; // TRUE时XY2-X导向电源通讯正常 
	PARAM040:REAL ; // XY2-Y导向电源电流设置值（A） 
	PARAM041:BOOL ; // XY2-Y导向电源已开 
	PARAM042:BOOL ; // XY2-Y导向电源已关 
	PARAM043:BOOL ; // XY2-Y导向电源正在开 
	PARAM044:BOOL ; // XY2-Y导向电源正在关 
	PARAM045:REAL ; // XY2-Y导向电源运行电流（A） 
	PARAM046:REAL ; // XY2-Y导向电源运行电压（V） 
	PARAM047:BOOL ; // TRUE时XY2-Y导向电源故障 
	PARAM048:BOOL ; // TRUE时XY2-Y导向电源电流操作错误 
	PARAM049:BOOL ; // TRUE时XY2-Y导向电源通讯正常 
	PARAM050:REAL ; // 螺旋管2电源电流设置值（A） 
	PARAM051:BOOL ; // 螺旋管2电源已开 
	PARAM052:BOOL ; // 螺旋管2电源已关 
	PARAM053:BOOL ; // 螺旋管2电源正在开 
	PARAM054:BOOL ; // 螺旋管2电源正在关 
	PARAM055:REAL ; // 螺旋管2电源运行电流（A） 
	PARAM056:REAL ; // 螺旋管2电源运行电压（V） 
	PARAM057:BOOL ; // TRUE时螺旋管2电源故障 
	PARAM058:BOOL ; // TRUE时螺旋管2电源电流操作错误 
	PARAM059:BOOL ; // 注入FC抑制偏压电源已开 
	PARAM060:BOOL ; // 注入FC抑制偏压电源已关 
	PARAM061:BOOL ; // 注入FC抑制偏压电源正在开 
	PARAM062:BOOL ; // 注入FC抑制偏压电源正在关 
	PARAM063:REAL ; // 注入FC抑制偏压电源运行电流（A） 
	PARAM064:REAL ; // 注入FC抑制偏压电源运行电压（V） 
	PARAM065:BOOL ; // Ture为注入FC抑制偏压电源故障 
	PARAM066:BOOL ; // Ture为注入FC抑制偏压电源远控 
	PARAM067:BOOL ; // 注入FC抑制偏压电源正极 
	PARAM068:BOOL ; // 注入FC抑制偏压电源负极 
	PARAM069:BOOL ; // 注入FC抑制偏压电源电压操作错误 

END_STRUCT
END_TYPE

// ---- DUTs/System_Status_Struct/S_ISPSValues_To_PC_Struct.TcDUT
TYPE S_ISPSValues_To_PC_Struct :
STRUCT
	PARAM000:BOOL  ; // 离子源电源系统自动运行，TRUE为开启 
	PARAM001:REAL  ; // 离子源高压电源电流设置值（mA） 
	PARAM002:REAL  ; // 离子源高压电源电压设置值（kV） 
	PARAM003:BOOL  ; // 离子源高压电源开到位 
	PARAM004:BOOL  ; // 离子源高压电源关到位 
	PARAM005:BOOL  ; // 离子源高压电源正在开 
	PARAM006:BOOL  ; // 离子源高压电源正在关 
	PARAM007:BOOL  ; // 离子源高压电源使能到位 
	PARAM008:BOOL  ; // 离子源高压电源停止使能到位 
	PARAM009:BOOL  ; // 离子源高压电源正在使能 
	PARAM010:BOOL  ; // 离子源高压电源正在停止使能 
	PARAM011:BOOL  ; // 离子源高压电源高压状态 
	PARAM012:BOOL  ; // 离子源高压电源故障状态 
	PARAM013:BOOL  ; // 离子源高压电源模式状态 
	PARAM014:BOOL  ; // 离子源高压电源开启操作错误 
	PARAM015:BOOL  ; // 离子源高压电源关闭操作错误 
	PARAM016:BOOL  ; // 离子源高压电源电流设置操作错误 
	PARAM017:BOOL  ; // 离子源高压电源电压设置操作错误 
	PARAM018:REAL  ; // 离子源高压电源电流（mA） 
	PARAM019:REAL  ; // 离子源高压电源电压（kV） 
	PARAM020:REAL  ; // 灯丝电源电流设置值（A） 
	PARAM021:REAL  ; // 灯丝电源电压设置值（V） 
	PARAM022:BOOL  ; // TRUE为灯丝电源就绪 
	PARAM023:BOOL  ; // 灯丝电源TRUE远控，FALSE本控 
	PARAM024:BOOL  ; // TRUE为灯丝电源故障 
	PARAM025:BOOL  ; // TRUE为灯丝电源过压 
	PARAM026:BOOL  ; // TRUE为灯丝电源过流 
	PARAM027:BOOL  ; // TRUE为灯丝电源过温 
	PARAM028:BOOL  ; // 灯丝电源外部连锁，TRUE正常 
	PARAM029:BOOL  ; // 灯丝电源已经运行 
	PARAM030:BOOL  ; // 灯丝电源停止运行 
	PARAM031:BOOL  ; // 灯丝电源正在启动运行 
	PARAM032:BOOL  ; // 灯丝电源正在停止运行 
	PARAM033:BOOL  ; // TRUE为灯丝电源控制器正常 
	PARAM034:BOOL  ; // 灯丝电源电流设置操作错误 
	PARAM035:BOOL  ; // 灯丝电源电压设置操作错误 
	PARAM036:REAL  ; // 灯丝电源运行电流（A） 
	PARAM037:REAL  ; // 灯丝电源运行电压（V） 
	PARAM038:REAL  ; // 弧压电源电流设置值（A） 
	PARAM039:REAL  ; // 弧压电源电压设置值（V） 
	PARAM040:BOOL  ; // TRUE为弧压电源就绪ON 
	PARAM041:BOOL  ; // 弧压电源TRUE远控，FALSE本控 
	PARAM042:BOOL  ; // TRUE为弧压电源故障 
	PARAM043:BOOL  ; // TRUE为弧压电源过压 
	PARAM044:BOOL  ; // TRUE为弧压电源过流 
	PARAM045:BOOL  ; // TRUE为弧压电源过温 
	PARAM046:BOOL  ; // 弧压电源外部连锁，TRUE正常 
	PARAM047:BOOL  ; // 弧压电源已经运行 
	PARAM048:BOOL  ; // 弧压电源停止运行 
	PARAM049:BOOL  ; // 弧压电源正在启动运行 
	PARAM050:BOOL  ; // 弧压电源正在停止运行 
	PARAM051:BOOL  ; // TRUE为弧压电源控制器正常
	PARAM052:BOOL  ; // 弧压电源电流设置操作错误 
	PARAM053:BOOL  ; // 弧压电源电压设置操作错误 
	PARAM054:REAL  ; // 弧压电源运行电流（A） 
	PARAM055:REAL  ; // 弧压电源运行电压（V） 
	PARAM056:REAL  ; // 等离子体电源电流设置值（A） 
	PARAM057:REAL  ; // 等离子体电源电压设置值（V） 
	PARAM058:BOOL  ; // TRUE为等离子体电源就绪ON 
	PARAM059:BOOL  ; // 等离子体电源TRUE远控，FALSE本控 
	PARAM060:BOOL  ; // TRUE为等离子体电源故障 
	PARAM061:BOOL  ; // TRUE为等离子体电源过压 
	PARAM062:BOOL  ; // TRUE为等离子体电源过流 
	PARAM063:BOOL  ; // TRUE为等离子体电源过温 
	PARAM064:BOOL  ; // 等离子体电源外部连锁，TRUE正常 
	PARAM065:BOOL  ; // 等离子体电源已经运行 
	PARAM066:BOOL  ; // 等离子体电源停止运行 
	PARAM067:BOOL  ; // 等离子体电源正在启动运行 
	PARAM068:BOOL  ; // 等离子体电源正在停止运行 
	PARAM069:BOOL  ; // TRUE为等离子体电源控制器正常 
	PARAM070:BOOL  ; // 等离子体电源电流设置操作错误 
	PARAM071:BOOL  ; // 等离子体电源电压设置操作错误 
	PARAM072:REAL  ; // 等离子体电源运行电流（A） 
	PARAM073:REAL  ; // 等离子体电源运行电压（V） 
	PARAM074:REAL  ; // 吸极电源电流设置值（A） 
	PARAM075:REAL  ; // 吸极电源电压设置值（V） 
	PARAM076:BOOL  ; // TRUE为吸极电源就绪ON 
	PARAM077:BOOL  ; // 吸极电源TRUE远控，FALSE本控 
	PARAM078:BOOL  ; // TRUE为吸极电源故障 
	PARAM079:BOOL  ; // TRUE为吸极电源过压 
	PARAM080:BOOL  ; // TRUE为吸极电源过流 
	PARAM081:BOOL  ; // TRUE为吸极电源过温 
	PARAM082:BOOL  ; // 吸极电源外部连锁，TRUE正常 
	PARAM083:BOOL  ; // 吸极电源已经运行 
	PARAM084:BOOL  ; // 吸极电源停止运行 
	PARAM085:BOOL  ; // 吸极电源正在启动运行 
	PARAM086:BOOL  ; // 吸极电源正在停止运行 
	PARAM087:BOOL  ; // TRUE为吸极电源控制器正常 
	PARAM088:BOOL  ; // 吸极电源电流设置操作错误 
	PARAM089:BOOL  ; // 吸极电源电压设置操作错误 
	PARAM090:REAL  ; // 吸极电源运行电流（A） 
	PARAM091:REAL  ; // 吸极电源运行电压（V）


END_STRUCT
END_TYPE

// ---- DUTs/System_Status_Struct/S_ISVacValues_To_PC_Struct.TcDUT
TYPE S_ISVacValues_To_PC_Struct :
STRUCT
	PARAM000:BOOL ; // 离子源低真空自动运行，True代表开 
	PARAM001:BOOL ; // 离子源高真空自动运行，True代表开 
	PARAM002:BOOL ; // 角阀2开到位
	PARAM003:BOOL ; // 角阀2关到位 
	PARAM004:BOOL ; // 角阀2正在开 
	PARAM005:BOOL ; // 角阀2正在关 
	PARAM006:BOOL ; // 角阀2开启操作错误 
	PARAM007:BOOL ; // 角阀2关闭操作错误 
	PARAM008:BOOL ; // 角阀3开到位 
	PARAM009:BOOL ; // 角阀3关到位 
	PARAM010:BOOL ; // 角阀3正在开 
	PARAM011:BOOL ; // 角阀3正在关 
	PARAM012:BOOL ; // 角阀3开启操作错误 
	PARAM013:BOOL ; // 角阀3关闭操作错误 
	PARAM014:BOOL ; // 注入线放气阀开到位 
	PARAM015:BOOL ; // 注入线放气阀关到位 
	PARAM016:BOOL ; // 注入线放气阀正在开 
	PARAM017:BOOL ; // 注入线放气阀正在关 
	PARAM018:BOOL ; // 注入线放气阀开启操作错误 
	PARAM019:BOOL ; // 注入线放气阀关闭操作错误 
	PARAM020:BOOL ; // 注入线干泵开到位 
	PARAM021:BOOL ; // 注入线干泵关到位 
	PARAM022:BOOL ; // 注入线干泵正在开 
	PARAM023:BOOL ; // 注入线干泵正在关 
	PARAM024:BOOL ; // 注入线干泵开启操作错误 
	PARAM025:BOOL ; // 注入线干泵关闭操作错误 
	PARAM026:BOOL ; // 分子泵V1达到频率值 
	PARAM027:BOOL ; // 分子泵V1频率下降到0 
	PARAM028:BOOL ; // 分子泵V1故障 
	PARAM029:BOOL ; // 分子泵V1频率上升中 
	PARAM030:BOOL ; // 分子泵V1频率下降中 
	PARAM031:BOOL ; // 分子泵V1开启操作错误 
	PARAM032:BOOL ; // 分子泵V1关闭操作错误 
	PARAM033:REAL ; // 分子泵V1输出频率（Hz）
	PARAM034:BOOL ; // 分子泵V3达到频率值 
	PARAM035:BOOL ; // 分子泵V3频率下降到0 
	PARAM036:BOOL ; // 分子泵V3故障 
	PARAM037:BOOL ; // 分子泵V3频率上升中 
	PARAM038:BOOL ; // 分子泵V3频率下降中 
	PARAM039:BOOL ; // 分子泵V3开启操作错误 
	PARAM040:BOOL ; // 分子泵V3关闭操作错误 
	PARAM041:REAL ; // 分子泵V3输出频率（Hz） 
	PARAM042:BOOL ; // 分子泵V4达到频率值 
	PARAM043:BOOL ; // 分子泵V4频率下降到0 
	PARAM044:BOOL ; // 分子泵V4故障 
	PARAM045:BOOL ; // 分子泵V4频率上升中 
	PARAM046:BOOL ; // 分子泵V4频率下降中 
	PARAM047:BOOL ; // 分子泵V4开启操作错误 
	PARAM048:BOOL ; // 分子泵V4关闭操作错误
	PARAM049:REAL ; // 分子泵V4输出频率（Hz） 
	PARAM050:LREAL ; // 离子源低真空度（mBar） 
	PARAM051:LREAL ; // 离子源高真空度（mBar） 
	PARAM052:BOOL ; // 离子源低真空达标 
	PARAM053:BOOL ; // 离子源高真空达标
END_STRUCT
END_TYPE

// ---- DUTs/System_Status_Struct/S_MainPSValues_To_PC_Struct.TcDUT
TYPE S_MainPSValues_To_PC_Struct :
STRUCT
	PARAM000:BOOL ; // 主器电源系统自动运行，TRUE为开启 
	PARAM001:REAL ; // 正偏转版电源电流设置值（mA） 
	PARAM002:REAL ; // 正偏转版电源电压设置值（kV） 
	PARAM003:BOOL ; // 正偏转版电源已开 
	PARAM004:BOOL ; // 正偏转版电源已关 
	PARAM005:BOOL ; // 正偏转版电源正在开 
	PARAM006:BOOL ; // 正偏转版电源正在关 
	PARAM007:BOOL ; // 正偏转版电源使能到位 
	PARAM008:BOOL ; // 正偏转版电源停止使能到位 
	PARAM009:BOOL ; // 正偏转版电源正在使能 
	PARAM010:BOOL ; // 正偏转版电源正在停止使能 
	PARAM011:BOOL ; // 正偏转版电源高压状态 
	PARAM012:BOOL ; // 正偏转版电源故障状态 
	PARAM013:BOOL ; // 正偏转版电源模式状态 
	PARAM014:BOOL ; // 正偏转版电源开启操作错误 
	PARAM015:BOOL ; // 正偏转版电源关闭操作错误 
	PARAM016:BOOL ; // 正偏转版电源电流设置操作错误 
	PARAM017:BOOL ; // 正偏转版电源电压设置操作错误
	PARAM018:REAL ; // 正偏转版电源电流（mA） 
	PARAM019:REAL ; // 正偏转版电源电压（kV） 
	PARAM020:REAL ; // 负偏转版电源电流设置值（mA） 
	PARAM021:REAL ; // 负偏转版电源电压设置值（kV） 
	PARAM022:BOOL ; // 负偏转版电源已开 
	PARAM023:BOOL ; // 负偏转版电源已关 
	PARAM024:BOOL ; // 负偏转版电源正在开 
	PARAM025:BOOL ; // 负偏转版电源正在关 
	PARAM026:BOOL ; // 负偏转版电源使能到位 
	PARAM027:BOOL ; // 负偏转版电源停止使能到位 
	PARAM028:BOOL ; // 负偏转版电源正在使能 
	PARAM029:BOOL ; // 负偏转版电源正在停止使能 
	PARAM030:BOOL ; // 负偏转版电源高压状态 
	PARAM031:BOOL ; // 负偏转版电源故障状态 
	PARAM032:BOOL ; // 负偏转版电源模式状态 
	PARAM033:BOOL ; // 负偏转版电源开启操作错误 
	PARAM034:BOOL ; // 负偏转版电源关闭操作错误 
	PARAM035:BOOL ; // 负偏转版电源电流设置操作错误 
	PARAM036:BOOL ; // 负偏转版电源电压设置操作错误 
	PARAM037:REAL ; // 负偏转版电源电流（mA） 
	PARAM038:REAL ; // 负偏转版电源电压（kV） 
	PARAM039:REAL ; // 主磁铁电源电流设置值（A） 
	PARAM040:BOOL ; // 主磁铁电源已开 
	PARAM041:BOOL ; // 主磁铁电源已关 
	PARAM042:BOOL ; // 主磁铁电源正在开 
	PARAM043:BOOL ; // 主磁铁电源正在关 
	PARAM044:REAL ; // 主磁铁电源运行电流（A） 
	PARAM045:REAL ; // 主磁铁电源运行电压（V） 
	PARAM046:BOOL ; // TRUE时主磁铁电源故障 
	PARAM047:BOOL ; // 主磁铁电源电流设置操作错误 
	PARAM048:REAL ; // 引出磁铁电源电流设置值（A） 
	PARAM049:BOOL ; // 引出磁铁电源已开 
	PARAM050:BOOL ; // 引出磁铁电源已关 
	PARAM051:BOOL ; // 引出磁铁电源正在开 
	PARAM052:BOOL ; // 引出磁铁电源正在关 
	PARAM053:REAL ; // 引出磁铁电源运行电流（A） 
	PARAM054:REAL ; // 引出磁铁电源运行电压（V） 
	PARAM055:BOOL ; // TRUE时引出磁铁电源故障 
	PARAM056:BOOL ; // 引出磁铁电源电流设置操作错误 
	PARAM057:BOOL ; // TRUE时引出磁铁电源通讯正常
END_STRUCT
END_TYPE

// ---- DUTs/System_Status_Struct/S_MainVacValues_To_PC_Struct.TcDUT
TYPE S_MainVacValues_To_PC_Struct :
STRUCT
	PARAM000:BOOL ; // 主真空低真空自动运行，True代表开 
	PARAM001:BOOL ; // 主真空高真空自动运行，True代表开 
	PARAM002:BOOL ; // 冷泵隔断阀1开到位 
	PARAM003:BOOL ; // 冷泵隔断阀1关到位 
	PARAM004:BOOL ; // 冷泵隔断阀1正在开 
	PARAM005:BOOL ; // 冷泵隔断阀1正在关 
	PARAM006:BOOL ; // 冷泵隔断阀1开启操作错误 
	PARAM007:BOOL ; // 冷泵隔断阀1关闭操作错误 
	PARAM008:BOOL ; // 冷泵隔断阀2开到位 
	PARAM009:BOOL ; // 冷泵隔断阀2关到位 
	PARAM010:BOOL ; // 冷泵隔断阀2正在开 
	PARAM011:BOOL ; // 冷泵隔断阀2正在关 
	PARAM012:BOOL ; // 冷泵隔断阀2开启操作错误 
	PARAM013:BOOL ; // 冷泵隔断阀2关闭操作错误 
	PARAM014:BOOL ; // 角阀1开到位 
	PARAM015:BOOL ; // 角阀1关到位 
	PARAM016:BOOL ; // 角阀1正在开 
	PARAM017:BOOL ; // 角阀1正在关 
	PARAM018:BOOL ; // 角阀1开启操作错误 
	PARAM019:BOOL ; // 角阀1关闭操作错误 
	PARAM020:BOOL ; // 主真空放气阀开到位 
	PARAM021:BOOL ; // 主真空放气阀关到位 
	PARAM022:BOOL ; // 主真空放气阀正在开 
	PARAM023:BOOL ; // 主真空放气阀正在关 
	PARAM024:BOOL ; // 主真空放气阀开启操作错误 
	PARAM025:BOOL ; // 主真空放气阀关闭操作错误
	PARAM026:BOOL ; // 主真空干泵开到位 
	PARAM027:BOOL ; // 主真空干泵关到位 
	PARAM028:BOOL ; // 主真空干泵正在开 
	PARAM029:BOOL ; // 主真空干泵正在关 
	PARAM030:BOOL ; // 主真空干泵开启操作错误 
	PARAM031:BOOL ; // 主真空干泵关闭操作错误 
	PARAM032:BOOL ; // 主真空分子泵V2达到频率值 
	PARAM033:BOOL ; // 主真空分子泵V2频率下降到0 
	PARAM034:BOOL ; // 主真空分子泵V2故障 
	PARAM035:BOOL ; // 主真空分子泵V2频率上升中 
	PARAM036:BOOL ; // 主真空分子泵V2频率下降中 
	PARAM037:BOOL ; // 主真空分子泵V2开启操作错误 
	PARAM038:BOOL ; // 主真空分子泵V2关闭操作错误 
	PARAM039:REAL ; // 主真空分子泵V2输出频率（Hz） 
	PARAM040:BOOL ; // 冷泵1前级阀开到位 
	PARAM041:BOOL ; // 冷泵1前级阀关到位 
	PARAM042:BOOL ; // 冷泵1前级阀正在开 
	PARAM043:BOOL ; // 冷泵1前级阀正在关 
	PARAM044:BOOL ; // 冷泵1前级阀通讯状态 
	PARAM045:BOOL ; // 冷泵1前级阀开启操作错误 
	PARAM046:BOOL ; // 冷泵1前级阀关闭操作错误 
	PARAM047:BOOL ; // 冷泵1开到位 
	PARAM048:BOOL ; // 冷泵1关到位 
	PARAM049:BOOL ; // 冷泵1正在开 
	PARAM050:BOOL ; // 冷泵1正在关 
	PARAM051:BOOL ; // 冷泵1通讯状态 
	PARAM052:REAL ; // 冷泵1一级冷板温度 
	PARAM053:REAL ; // 冷泵1二级冷板温度
	PARAM054:REAL ; // 冷泵1真空度 
	PARAM055:BOOL ; // 冷泵1开启操作错误 
	PARAM056:BOOL ; // 冷泵1关闭操作错误 
	PARAM057:BOOL ; // 冷泵2前级阀开到位 
	PARAM058:BOOL ; // 冷泵2前级阀关到位 
	PARAM059:BOOL ; // 冷泵2前级阀正在开 
	PARAM060:BOOL ; // 冷泵2前级阀正在关 
	PARAM061:BOOL ; // 冷泵2前级阀通讯状态 
	PARAM062:BOOL ; // 冷泵2前级阀开启操作错误 
	PARAM063:BOOL ; // 冷泵2前级阀关闭操作错误 
	PARAM064:BOOL ; // 冷泵2开到位 
	PARAM065:BOOL ; // 冷泵2关到位 
	PARAM066:BOOL ; // 冷泵2正在开 
	PARAM067:BOOL ; // 冷泵2正在关 
	PARAM068:BOOL ; // 冷泵2通讯状态 
	PARAM069:REAL ; // 冷泵2一级冷板温度 
	PARAM070:REAL ; // 冷泵2二级冷板温度 
	PARAM071:REAL ; // 冷泵2真空度 
	PARAM072:BOOL ; // 冷泵2开启操作错误 
	PARAM073:BOOL ; // 冷泵2关闭操作错误 
	PARAM074:LREAL ; //  主真空低真空度（mBar） 
	PARAM075:LREAL ; //  主真空高真空度（mBar） 
	PARAM076:BOOL ; // 主真空低真空达标 
	PARAM077:BOOL ; // 主真空高真空达标
	

END_STRUCT
END_TYPE

// ---- DUTs/System_Status_Struct/S_RFValues_To_PC_Struct.TcDUT
TYPE S_RFValues_To_PC_Struct :
STRUCT
	PARAM000:BOOL ;// 高频发射机1已上电 
	PARAM001:BOOL ;// 高频发射机1已停电 
	PARAM002:BOOL ;// 高频发射机1正在上电 
	PARAM003:BOOL ;// 高频发射机1正在停电 
	PARAM004:BOOL ;// 高频发射机1高压已上电 
	PARAM005:BOOL ;// 高频发射机1高压已停电 
	PARAM006:BOOL ;// 高频发射机1高压正在上电 
	PARAM007:BOOL ;// 高频发射机1高压正在停电 
	PARAM008:BOOL ;// 高频发射机1风冷状态 
	PARAM009:BOOL ;// 高频发射机1水冷状态 
	PARAM010:BOOL ;// 高频发射机1主变压器温度 
	PARAM011:BOOL ;// 高频发射机1门开关 
	PARAM012:BOOL ;// 高频发射机1冷却加电完成 
	PARAM013:BOOL ;// 高频发射机1灯丝加电完成 
	PARAM014:BOOL ;// 高频发射机1固态加电完成 
	PARAM015:BOOL ;// 高频发射机1高压加电完成 
	PARAM016:BOOL ;// 高频发射机1风冷状态锁存 
	PARAM017:BOOL ;// 高频发射机1水冷状态锁存 
	PARAM018:BOOL ;// 高频发射机1主变压器温度锁存 
	PARAM019:BOOL ;// 高频发射机1门开关锁存 
	PARAM020:BOOL ;// 高频发射机1外部连锁锁存 
	PARAM021:BOOL ;// 高频发射机1阳极过流锁存 
	PARAM022:BOOL ;// 高频发射机1反射过大锁存 
	PARAM023:BOOL ;// 高频发射机1冷却汇总锁存 
	PARAM024:BOOL ;// 高频发射机1闭锁汇总锁存 
	PARAM025:BOOL ;// 高频发射机1过荷汇总锁存 
	PARAM026:BOOL ;// 高频发射机1冷却汇总 
	PARAM027:BOOL ;// 高频发射机1闭锁汇总 
	PARAM028:BOOL ;// 高频发射机1过荷汇总 
	PARAM029:REAL ;// 高频发射机1灯丝电流 
	PARAM030:REAL ;// 高频发射机1栅极电流 
	PARAM031:REAL ;// 高频发射机1阳极电压 
	PARAM032:REAL ;// 高频发射机1阳极电流 
	PARAM033:REAL ;// 高频发射机1入射功率 
	PARAM034:REAL ;// 高频发射机1反射功率 
	PARAM035:BOOL ;// 高频发射机2已上电 
	PARAM036:BOOL ;// 高频发射机2已停电 
	PARAM037:BOOL ;// 高频发射机2正在上电 
	PARAM038:BOOL ;// 高频发射机2正在停电 
	PARAM039:BOOL ;// 高频发射机2高压已上电 
	PARAM040:BOOL ;// 高频发射机2高压已停电 
	PARAM041:BOOL ;// 高频发射机2高压正在上电 
	PARAM042:BOOL ;// 高频发射机2高压正在停电 
	PARAM043:BOOL ;// 高频发射机2风冷状态 
	PARAM044:BOOL ;// 高频发射机2水冷状态 
	PARAM045:BOOL ;// 高频发射机2主变压器温度 
	PARAM046:BOOL ;// 高频发射机2门开关 
	PARAM047:BOOL ;// 高频发射机2冷却加电完成 
	PARAM048:BOOL ;// 高频发射机2灯丝加电完成 
	PARAM049:BOOL ;// 高频发射机2固态加电完成 
	PARAM050:BOOL ;// 高频发射机2高压加电完成
	PARAM051:BOOL ;// 高频发射机2风冷状态锁存 
	PARAM052:BOOL ;// 高频发射机2水冷状态锁存 
	PARAM053:BOOL ;// 高频发射机2主变压器温度锁存 
	PARAM054:BOOL ;// 高频发射机2门开关锁存 
	PARAM055:BOOL ;// 高频发射机2外部连锁锁存 
	PARAM056:BOOL ;// 高频发射机2阳极过流锁存 
	PARAM057:BOOL ;// 高频发射机2反射过大锁存 
	PARAM058:BOOL ;// 高频发射机2冷却汇总锁存 
	PARAM059:BOOL ;// 高频发射机2闭锁汇总锁存 
	PARAM060:BOOL ;// 高频发射机2过荷汇总锁存 
	PARAM061:BOOL ;// 高频发射机2冷却汇总 
	PARAM062:BOOL ;// 高频发射机2闭锁汇总 
	PARAM063:BOOL ;// 高频发射机2过荷汇总 
	PARAM064:REAL ;// 高频发射机2灯丝电流 
	PARAM065:REAL ;// 高频发射机2栅极电流 
	PARAM066:REAL ;// 高频发射机2阳极电压 
	PARAM067:REAL ;// 高频发射机2阳极电流 
	PARAM068:REAL ;// 高频发射机2入射功率 
	PARAM069:REAL ;// 高频发射机2反射功率 
	

END_STRUCT
END_TYPE

// ---- DUTs/System_Status_Struct/S_WCValues_To_PC_Struct.TcDUT
TYPE S_WCValues_To_PC_Struct :
STRUCT
	PARAM000:BOOL ; // 主器水流继电器 01 高频上 1#
	PARAM001:BOOL ; // 主器水流继电器 02 高频上 2#
	PARAM002:BOOL ; // 主器水流继电器 03 高频下 1#
	PARAM003:BOOL ; // 主器水流继电器 04 高频下 2#
	PARAM004:BOOL ; // 主器水流继电器 05 上线圈
	PARAM005:BOOL ; // 主器水流继电器 06 下线圈
	PARAM006:BOOL ; // 主器水流继电器 07 聚束器分路
	PARAM007:BOOL ; // 主器水流继电器 08 离子源
	PARAM008:BOOL ; // 主器水流继电器 09 内靶
	PARAM009:BOOL ; // 主器水流继电器 10 螺旋管
	PARAM010:BOOL ; // 主器水流继电器 11 冷泵
	PARAM011:BOOL ; // 主器水流继电器 12 主真空
	PARAM012:BOOL ; // 主器水流继电器 13 离子源分支
	PARAM013:BOOL ; // 主器水流继电器 14 备用
	PARAM014:BOOL ; // 束流线水流继电器 01
	PARAM015:BOOL ; // 束流线水流继电器 02
	PARAM016:BOOL ; // 束流线水流继电器 03
	PARAM017:BOOL ; // 束流线水流继电器 04
	PARAM018:BOOL ; // 束流线水流继电器 05
	PARAM019:BOOL ; // 束流线水流继电器 06
	PARAM020:BOOL ; // 束流线水流继电器 07
	PARAM021:BOOL ; // 束流线水流继电器 08
END_STRUCT
END_TYPE

// ---- DUTs/ST_FrameCmd.TcDUT
TYPE ST_FrameCmd :
STRUCT
	sys   : BYTE;
    sub_s : BYTE;
    dev   : BYTE;
    cmd   : BYTE;
    set   : REAL;
END_STRUCT
END_TYPE

// ---- DUTs/System_Status_Struct/TCSSys_Struct.TcDUT
TYPE TCSSys_Struct :
STRUCT
	PARAM000:BOOL ;// 只读，TRUE为加速器准备好
	PARAM001:BOOL ;// 读写，TRUE为TCS准备好  
	PARAM002:BOOL ;// 只读，TRUE代表加速器出束 
	PARAM003:BOOL ;// 读写，TRUE为TCS系统正在运行  
END_STRUCT
END_TYPE

// ---- POUs/MAIN.TcPOU
PROGRAM MAIN
VAR
	Framecmd:ST_FrameCmd;
	CommandExcute:BOOL;
	TEST1:UINT;
TEST2:UINT;
TEST3:UINT;
TEST4:UINT;
TEST5:UINT;
TEST6:UINT;
TEST7:UINT;
TEST8:UINT;
TEST9:UINT;
TEST10:UINT;
TEST11:UINT;
TEST12:UINT;
TEST13:UINT;
TEST14:UINT;
TEST15:UINT;
END_VAR

TEST1 :=SIZEOF(S_WCValues_To_PC_Struct);
TEST2:=SIZEOF(S_ARValues_To_PC_Struct);
TEST3:=SIZEOF(S_ISVacValues_To_PC_Struct);
TEST4:=SIZEOF(S_MainVacValues_To_PC_Struct);
TEST5:=SIZEOF(S_BLVac1Values_To_PC_Struct);
TEST6:=SIZEOF(S_BLVac2Values_To_PC_Struct);
TEST7:=SIZEOF(S_BLVac3Values_To_PC_Struct);
TEST8:=SIZEOF(S_ISPSValues_To_PC_Struct);
TEST9:=SIZEOF(S_INJLPSValues_To_PC_Struct);
TEST10:=SIZEOF(S_MainPSValues_To_PC_Struct);
TEST11:=SIZEOF(S_BLPS1Values_To_PC_Struct);
TEST12:=SIZEOF(S_BLPS3Values_To_PC_Struct);
TEST13:=SIZEOF(S_RFValues_To_PC_Struct);
TEST14:=SIZEOF(S_BDValues_To_PC_Struct);
TEST15:=SIZEOF(S_ILValues_To_PC_Struct);

END_PROGRAM

// ---- POUs/Call_Values_To_PC.TcPOU
PROGRAM Call_Values_To_PC
VAR
	Read_WC_Values_To_PC:READ_WC_Values_To_PC_Struct; //3.4.1水冷系统
	Read_AR_Values_To_PC:Read_AR_Values_To_PC_Struct; //3.4.2气动系统
	Read_ISVac_Values_To_PC:Read_ISVac_Values_To_PC_Struct; //3.4.3离子源真空系统
	Read_MainVac_Values_To_PC:Read_MainVac_Values_To_PC_Struct; //3.4.4主真空系统
	Read_BLVac1_Values_To_PC:Read_BLVac1_Values_To_PC_Struct; //3.4.5 束流线 1（公共束流线）真空系统
	Read_BLVac2_Values_To_PC:Read_BLVac2_Values_To_PC_Struct; //3.4.6 束流线 2（公共束流线）真空系统
	Read_BLVac3_Values_To_PC:Read_BLVac3_Values_To_PC_Struct; //3.4.7 束流线 3（公共束流线）真空系统
	Read_ISPS_Values_To_PC:Read_ISPS_Values_To_PC_Struct; //3.4.8 离子源电源系统 
	Read_INJLPS_Values_To_PC:Read_INJLPS_Values_To_PC_Struct; //3.4.9 注入线电源系统
	Read_MainPS_Values_To_PC:Read_MainPS_Values_To_PC_Struct;  //3.4.10 主器电源系统
	Read_BLPS1_Values_To_PC:Read_BLPS1_Values_To_PC_Struct; //3.4.11 束流线 1（公共束流线）电源系统
	Read_BLPS3_Values_To_PC:Read_BLPS3_Values_To_PC_Struct; //3.4.12 束流线 3（中子靶束流线）电源系统
	Read_RFG_Values_To_PC:Read_RFG_Values_To_PC_Struct; //3.4.13 高频系统 
	Read_BD_Values_To_PC:Read_BD_Values_To_PC_Struct; //3.4.14 束流测量系统 
	Read_IL_Values_To_PC:Read_IL_Values_To_PC_Struct; //3.4.15 联锁系统
END_VAR

END_PROGRAM

// ---- POUs/Com_StripperEleMach.TcPOU
PROGRAM Com_StripperEleMach
VAR
	bEM_C_Power_Axis1        : BOOL;
	fEM_C_AbPos_Axis1        : REAL;
    fEM_C_AbPosVelo_Axis1    : REAL;
    bEM_C_AbPosExecute_Axis1 : BOOL;
    bEM_C_Reset_Axis1        : BOOL;
	bEM_C_Power_Axis2        : BOOL;
	fEM_C_AbPos_Axis2        : REAL;
    fEM_C_AbPosVelo_Axis2    : REAL;
    bEM_C_AbPosExecute_Axis2 : BOOL;
    bEM_C_Reset_Axis2        : BOOL;
END_VAR

END_PROGRAM

// ---- POUs/GVL_TCSSys.TcPOU
PROGRAM GVL_TCSSys
VAR
	TCSSys:TCSSys_Struct; //3.4.16 TCS系统
END_VAR

END_PROGRAM
